{attribute 'qualified_only'}
{attribute 'strict'}
TYPE E_LaudaParameterWriteState :
(
	READY,
	SEND,
	AWAIT_RESPONSE,
	VALIDATE_RESPONSE,
	DONE
);
END_TYPE

(* stored: Version 1.1.0.1, ProductVersion 3.1.4024.13
   DUT E_LaudaParameterWriteState: Id {2d063000-6fc6-0f7b-368d-d0fc2af3fc45} *)
